# B&R Automation Studio project Sew
Automation Studio 4.12.2.93

## Configuration Config1

CPU PC_any, AutomationRuntime B4.93, Build 4.1.2, Vc V4.72.7

### Hardware
```
PC : PC_any v1.1.1.0 (OrderNumber=PC)
```

## Logical view

### Program Logical/Program

#### Main.st
```iecst
PROGRAM _INIT
	(* Insert code here *)

END_PROGRAM

PROGRAM _CYCLIC
	(* Insert code here *)
	IF expression THEN

	END_IF;
END_PROGRAM

PROGRAM _EXIT
	(* Insert code here *)

END_PROGRAM
```
